// TIA Portal V19 export
DATA_BLOCK "DB_HMI Support"   // DB10000
{ S7_Optimized_Access := 'FALSE' }
// stored: AutoNumber false
   VAR
      "PLC Mode" : Int;
      "PLC Near Status" : Int;
      "PLC Far Status" : Int;
      "Bypasses Status" : Int;
      OperationStateSystem : Int;
      MRPRingState : Int;
   END_VAR
BEGIN
END_DATA_BLOCK
